FUNCTION_BLOCK AUI_TO_AR (* Composite FB for converting AUI (UINT) adapter to AR (REAL) adapter — numeric conversion (value-preserving cast; narrowing may truncate, widening/sign-extension is safe). *)
  (* Standard: 61499-2; Description: Copyright (c) 2026 HR Agrartechnik GmbH This program and the accompanying materials are made available under the terms of the Eclipse Public License 2.0 which is available at https://www.eclipse.org/legal/epl-2.0/ SPDX-License-Identifier: EPL-2.0 *)
  (* Version 1.0, 2026-02-17, Franz Höpfinger, HR Agrartechnik GmbH *)
  PACKAGE adapter::conversion::unidirectional;
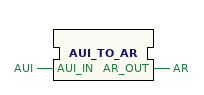
  SOCKETS
    AUI_IN : adapter::types::unidirectional::AUI; (* UINT Adapter Input *)
  END_SOCKETS
  PLUGS
    AR_OUT : adapter::types::unidirectional::AR; (* REAL Adapter Output *)
  END_PLUGS
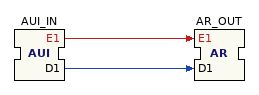
  EVENT_CONNECTIONS
    AUI_IN.E1 TO AR_OUT.E1;
  END_CONNECTIONS
  DATA_CONNECTIONS
    AUI_IN.D1 TO AR_OUT.D1;
  END_CONNECTIONS
END_FUNCTION_BLOCK
